Staubli VAL3: bindRow.pgx

public program bindRow()
begin
end
